FUNCTION_BLOCK INTERNAL FB_HasInstanceName_Tests EXTENDS FB_TestSuite
VAR_INPUT
END_VAR
VAR_OUTPUT
END_VAR
VAR
	fbHasInstanceName	:  FB_HasInstanceName_ExtensionForTests;
END_VAR

Test01_InstanceName();
Test02_InstancePath();

METHOD Test01_InstanceName
VAR_INPUT
END_VAR
TcUnit.TEST('Test01_InstanceName');

AssertEquals_STRING(
	Expected := 'fbHasInstanceName',
	Actual := fbHasInstanceName.InstanceName,
	Message := 'InstanceName is not correct.');
	
TcUnit.TEST_FINISHED();
END_METHOD

METHOD Test02_InstancePath
VAR_INPUT
END_VAR
TcUnit.TEST('Test02_InstancePath');

AssertEquals_STRING(
	Expected := 'PRG_TESTS.HasInstanceNameTests.fbHasInstanceName',
	Actual := fbHasInstanceName.InstancePath,
	Message := 'Instance path is incorrect.');

TcUnit.TEST_FINISHED();
END_METHOD

END_FUNCTION_BLOCK

(* stored: Version 1.1.0.1, ProductVersion 3.1.4024.14
   POU FB_HasInstanceName_Tests: Id {fc7f1c45-4e05-0854-19c6-d70a4b102dae}, SpecialFunc None
   Method Test01_InstanceName: Id {5d7d088d-abcc-0fd9-2182-97fbd3514b3d}
   Method Test02_InstancePath: Id {f581677f-1ea9-0956-3189-c0c8eb6c191a} *)
